// TIA Portal V17 export
// export: Created 2024-08-20T13:26:12.9911753Z, ExportSetting WithDefaults, DisplayName Totally Integrated Automation Portal, DisplayVersion V17 Update 4, DisplayName TIA Portal Openness, DisplayVersion V17 Update 4, DisplayName TIA Portal Version Control Interface, DisplayVersion V17, DisplayName STEP 7 Professional, DisplayVersion V17 Update 4, DisplayName STEP 7 Safety, DisplayVersion V17, DisplayName WinCC Advanced, DisplayVersion V17 Update 4
VAR_GLOBAL   // PLC tag table "ALARMES"
   ALM0 AT %MW100 : Word;   // ALARMES MB-01
   ALM2 AT %MW102 : Word;   // ALARMES MB-02
   ALM4 AT %MW104 : Word;   // ALARMES MB-03
   ALM6 AT %MW106 : Word;   // ALARMES MB-04
   ALM8 AT %MW108 : Word;   // ALARMES LIT_001
   ALM10 AT %MW110 : Word;   // ALARMES PCM-EEE
   ALM12 AT %MW112 : Word;   // ALARMES QGBT
   ALM14 AT %MW114 : Word;   // ALARMES CHAVE DE NIVEL
   ALM16 AT %MW116 : Word;   // ALARMES PCE-EEE
END_VAR
